// TwinCAT 3 PLC project MAS418
// ProgramVersion: 3.1.4023.0
// libraries:
//   Tc2_Standard, * (Beckhoff Automation GmbH)
//   Tc2_System, * (Beckhoff Automation GmbH)
//   Tc3_Module, * (Beckhoff Automation GmbH)
// project tree:
//   ControlBox/ CL_PC.TcPOU, E_Control_Mode.TcDUT, E_Status.TcDUT, FB_Connect.TcPOU, FB_ControlBox.TcPOU, FB_Encoder.TcPOU, FB_JoystickInputScaling.TcPOU, FB_PathGenerator.TcPOU, FB_Real_Controller.TcPOU, FB_ValveOutput.TcPOU, FB_Virtual_Controller.TcPOU, I_ControlBox.TcIO, OL_VC.TcPOU, ST_Control_Box.TcDUT, ST_ValveDeadBand.TcDUT (not stored)
//   ControlBox/GVL/ G_ControlBox.TcGVL, G_HMI.TcGVL, G_Input.TcGVL (not stored), G_IO_Parameters.TcGVL, G_Output.TcGVL, G_PathGen.TcGVL, G_Sim.TcGVL (not stored)
//   / GlobalTextList.TcGTLO, PlcTask.TcTTO, Visualization Manager.TcVMO (not stored)
//   HMI/ Visualization.TcVIS
//   Programs/FunctionBlock/ FB_Scaling.TcPOU
//   Programs/Functions/ F_NormFlow.TcPOU, F_Scaling.TcPOU, F_Hestunger.TcPOU
//   Programs/ MAIN.TcPOU, P_ControlBox.TcPOU
// real-time tasks:
//   TASK PlcTask: cycle T#10ms, priority 20, ADS port 350
// I/O:
//   DEVICE PLC (disabled), AmsNetId 192.168.56.1.2.1
//     Term 1 (EK1200) [EK1200-5000 EtherCAT Power supply (2A E-Bus)]
//       Term 2 (EL2008-0015) [EL2008-0015 8Ch. Dig. Output 24V DC, 0.35A, not short-circuit proof]
//       Term 3 (EL9011) [EL9011 End Terminal]
//   DEVICE Device 4 (EtherCAT), AmsNetId 5.80.90.242.5.1
//     Term 4 (EK1100) [EK1100 EtherCAT Coupler (2A E-Bus)]
//       DI1 (EL1008) [EL1008 8Ch. Dig. Input 24V, 3ms]
//       DO1 (EL2008)
//       AI1 (EL3068) [EL3068 8Ch. Ana. Input 0-10V]
//       AI2 (EL3068)
//       AI3 ( EL3174)
//       AI4  (EL3255) [EL3255 5Ch. potentiometer measurement with sensor supply]
//       AO1 (EL4104) [EL4104 4Ch. Ana. Output 0-10V, 16bit]
//       Term 10 (EL9011)
//     Encoder [Absolute Rotary Encoder IXARC V01.05]
// variable links:
//   MAS418 Instance <-> Device 4 (EtherCAT)/Encoder
//     PlcTask Inputs/G_Input.n_WinchEncoder <-> Encoder/Position Value
//   MAS418 Instance <-> Device 4 (EtherCAT)/Term 4 (EK1100)/AI1 (EL3068)
//     PlcTask Inputs/G_Input.n_pCA <-> AI Standard Channel 4/Value
//     PlcTask Inputs/G_Input.n_pCB <-> AI Standard Channel 3/Value
//     PlcTask Inputs/G_Input.n_pR <-> AI Standard Channel 2/Value
//     PlcTask Inputs/G_Input.n_pS <-> AI Standard Channel 1/Value
//     PlcTask Inputs/G_Input.n_pWA <-> AI Standard Channel 7/Value
//     PlcTask Inputs/G_Input.n_pWA1 <-> AI Standard Channel 5/Value
//     PlcTask Inputs/G_Input.n_pWB <-> AI Standard Channel 8/Value
//     PlcTask Inputs/G_Input.n_pWB1 <-> AI Standard Channel 6/Value
//   MAS418 Instance <-> Device 4 (EtherCAT)/Term 4 (EK1100)/AI2 (EL3068)
//     PlcTask Inputs/G_Input.n_pWD <-> AI Standard Channel 1/Value
//   MAS418 Instance <-> Device 4 (EtherCAT)/Term 4 (EK1100)/AI3 ( EL3174)
//     PlcTask Inputs/G_Input.n_QW <-> AI Standard Channel 1/Value
//   MAS418 Instance <-> Device 4 (EtherCAT)/Term 4 (EK1100)/AI4  (EL3255)
//     PlcTask Inputs/G_Input.n_JoyX <-> AI Standard Channel 2/Value
//     PlcTask Inputs/G_Input.n_JoyY <-> AI Standard Channel 3/Value
//     PlcTask Inputs/G_Input.n_Xc <-> AI Standard Channel 1/Value
//   MAS418 Instance <-> Device 4 (EtherCAT)/Term 4 (EK1100)/AO1 (EL4104)
//     PlcTask Outputs/G_Output.n_CylValveOut <-> AO Output Channel 2/Analog output
//     PlcTask Outputs/G_Output.n_WinchValveOut <-> AO Output Channel 1/Analog output
//   MAS418 Instance <-> Device 4 (EtherCAT)/Term 4 (EK1100)/DI1 (EL1008)
//     PlcTask Inputs/G_Input.bAuto <-> Channel 2/Input
//     PlcTask Inputs/G_Input.bJoyActive <-> Channel 5/Input
//     PlcTask Inputs/G_Input.bManual <-> Channel 1/Input
//     PlcTask Inputs/G_Input.bStart <-> Channel 3/Input
//     PlcTask Inputs/G_Input.bStop <-> Channel 4/Input
//   MAS418 Instance <-> Device 4 (EtherCAT)/Term 4 (EK1100)/DO1 (EL2008)
//     PlcTask Outputs/G_Output.bEnableCylValve <-> Channel 4/Output
//     PlcTask Outputs/G_Output.bEnableWinchValve <-> Channel 3/Output
//     PlcTask Outputs/G_Output.bGreenLED <-> Channel 1/Output
//     PlcTask Outputs/G_Output.bRedLED <-> Channel 2/Output

CONFIGURATION MAS418
    RESOURCE PLC ON TwinCAT3
        TASK PlcTask(INTERVAL := T#10ms, PRIORITY := 20);
        PROGRAM MAIN WITH PlcTask : MAIN;
    END_RESOURCE
END_CONFIGURATION

// ---- ControlBox/E_Control_Mode.TcDUT
{attribute 'qualified_only'}
{attribute 'strict'}
TYPE E_Control_Mode :
(
	OFF := 0,
	MANUAL := 1,
	AUTO := 2
);
END_TYPE

// ---- ControlBox/E_Status.TcDUT
{attribute 'qualified_only'}
{attribute 'strict'}
TYPE E_Status :
(
	NOTREADY,
	READY,
	STARTING,
	RUNNING,
	STOPPING,
	FAULT
);
END_TYPE

// ---- ControlBox/ST_Control_Box.TcDUT
TYPE ST_Control_Box :
STRUCT
	// Control mode variables
	eMode : E_Control_Mode; // Control mode for the control box
	bAuto : BOOL := FALSE; // Auto control mode input
	bManual : BOOL := FALSE; // Manual control mode input

	// Start/stop variables
	bStart : BOOL := FALSE; // Start button input
	bStop : BOOL := FALSE; // Stop button input

	// Joy variables
	bJoyActive : BOOL; // Activate the joystick boolean (Top switch)
	bJoyNotActive: BOOL; // Inverse logic of JoyActive
	fJoyX : REAL := 0; // Variable for storing the joy value in x direction (Cylinder)
	fJoyY : REAL := 0; // Variable for storing the joy value in y direction (Winch)
END_STRUCT
END_TYPE

// ---- ControlBox/GVL/G_ControlBox.TcGVL
VAR_GLOBAL
	// Global variable for control mode
	eMode : E_Control_Mode := E_Control_Mode.OFF;
	
	// GLobal variable for machine status
	eStatus : E_Status := E_Status.NOTREADY;
	
	// Timer between STARTING -> RUNNING and STOPPING -> NOTREADY
	fbTon : TON := ();
	bStartTimer : BOOL := FALSE;
	bTimerDone : BOOL;
	
	bStart : BOOL := FALSE; // Start button input
	bStop : BOOL := FALSE; // Stop button input
	
	bAuto : BOOL := FALSE; // Auto control mode input
	bManual : BOOL := FALSE; // Manual control mode input
	bOff : BOOL := FALSE; // Off mode
	
	bReady : BOOL := FALSE;
	bStarting : BOOL := FALSE;
	bRunning : BOOL := FALSE;
	bStopping : BOOL := FALSE;
	bFault : BOOL := FALSE;
	
	bJoyActive : BOOL; // Activate the joystick boolean (Top switch)
	bJoyNotActive: BOOL; // Inverse logic of JoyActive
	fJoyX : REAL := G_IO_Parameters.fMaxInputValue/2 + G_IO_Parameters.fMinInputValue/2; // Variable for storing the joy value in x direction (Cylinder)
	fJoyY : REAL := G_IO_Parameters.fMaxInputValue/2 + G_IO_Parameters.fMinInputValue/2; // Variable for storing the joy value in y direction (Winch)
	
	// Normalized values between -1 and 1
	fJoyX_Normalized : LREAL;
	fJoyY_Normalized : LREAL;
	
	// Open-Loop Velocity manual mode
	f_uVFF_winch_manual : LREAL;
	f_uVFF_cyl_manual : LREAL;
	
	// Closed-Loop auto mode
	f_uVFF_winch_auto : LREAL;
	f_uVFF_cyl_auto : LREAL;

	f_uPFB_winch_auto : LREAL;
	f_uPFB_cyl_auto : LREAL;
	
	f_u_winch : LREAL; // Summed winch control signal
	f_u_cyl : LREAL; // Summed cylinder control signal
	
	// Proportional gain
	fPGain : LREAL := 1;
	
	// Position feedback variable
	fPositionFeedback_winch : LREAL := 0;
	fPositionFeedback_cyl : LREAL := 0;
	
	fLimitVal : LREAL := 0.05;
END_VAR

// ---- ControlBox/GVL/G_HMI.TcGVL
VAR_GLOBAL	
	
	// inputs
	f_pS : REAL;
	f_pR : REAL;
	f_pCB : REAL;
	f_pCA : REAL;
	f_pWA1 : REAL;
	f_pWB1 : REAL;
	f_pWA: REAL;
	f_pWB : REAL;
	f_pWD : REAL;
	f_QW : REAL;
	f_Xc : REAL;
	f_JoyX : REAL;
	f_JoyY : REAL;
	f_WinchEncoder : LREAL;
	
END_VAR

// ---- ControlBox/GVL/G_IO_Parameters.TcGVL
{attribute 'qualified_only'}
VAR_GLOBAL
	// Joystick parameters
	fMaxInputValue : REAL := 20509.0;
	fMinInputValue : REAL := 11787.0;
	fNeutralInputValue : REAL := 16175;
	fNeutralDeadband : REAL := 50.0;
	fMaxOutputValue  : REAL := 1.0;
	fMinOutputValue : REAL := -1.0;
	fNeutralOutputValue : REAL := 0.0;
	
	// Deadband
	fPosMax : REAL := 29490.0;
	fPosMin : REAL := 20950.0;
	fNegMin : REAL := 18250.0;
	fNegMax : REAL := 9830.0;
	
	fMaxVel : LREAL := 0.05;
	
	fQmax_winch : LREAL := 60/60000; // L/min
	fQmax_cyl : LREAL := 75/60000; // L/min
END_VAR

// ---- ControlBox/GVL/G_Output.TcGVL
VAR_GLOBAL
	// Boolean outputs
	bGreenLED AT %Q* : BOOL;
	bRedLED AT %Q* : BOOL;
	bEnableWinchValve AT %Q* : BOOL;
	bEnableCylValve AT %Q* : BOOL;
	
	// DINT outputs
	n_WinchValveOut AT %Q* : DINT;
	n_CylValveOut AT %Q* : DINT;
END_VAR

// ---- ControlBox/GVL/G_PathGen.TcGVL
VAR_GLOBAL
	Enable : LREAL;
	x0 :LREAL := 0;  // [m], set at start
	x0_winch : LREAL := 0;
	x0_cyl : LREAL := 0;
	v0 :LREAL := 0; // [m/s], set at start
	Position_SP : LREAL := 0.1+x0; // [m], destination point. needs to set with logic. x + x0
	Velocity_SP : LREAL := 0.05*0.3; // [m/s], desired speed
	t0 : LREAL := 5.5; //[s], time to start ramp
	tRamp : LREAL := 1; // [s] ramp time (rise time)
	tHoldPos : LREAL := 1; // [s], time to stay at position before returning
	tVaiable : TIME := T#0S; // Time rising avfter timer is enabled
	tPT : TIME := T#200S; // Stop time for timer. Nessesery to work
	tQ : BOOL; // Gets true when stop time for timer is reached
	tStart : BOOL := FALSE; // enable to start timer. Rising edge start, falling reset
	fTime : LREAL;
	
	// OUTPUTS:
	fPositionRef : LREAL;
	fVelocityRef : LREAL;
	fTimeTot : LREAL; //Time needed to to the complete path
	fError : LREAL; // Should be changed to a BOOL
// SimulationTime is 
END_VAR

// ---- ControlBox/I_ControlBox.TcIO
INTERFACE I_ControlBox

METHOD Joy_Normalized : REAL
VAR_INPUT
	// Joy X
	fJoyX_raw : LREAL;
	// Joy Y
	fJoyY_raw : LREAL;
	
	// Min/max in/out parameters
	fMin_in : LREAL;
	fMax_in : LREAL;
	fMin_out : REAL;
	fMax_out : LREAL;
END_VAR
VAR_OUTPUT
	fJoyX_normalized : LREAL;
	fJoyY_normalized : LREAL;
END_VAR
END_METHOD

METHOD Mode
END_METHOD

METHOD Status
END_METHOD

END_INTERFACE

// ---- Programs/MAIN.TcPOU
PROGRAM MAIN
VAR
	fbScaling : FB_Scaling;
END_VAR

P_ControlBox(); // Run selected control box mode (virtual or real)
fbScaling();

END_PROGRAM

// ---- Programs/FunctionBlock/FB_Scaling.TcPOU
FUNCTION_BLOCK FB_Scaling
VAR
	fbEncoder : FB_Encoder();
	fbValveOutput : FB_ValveOutput();
END_VAR


//Test OK
F_NormFlow(nInput:= G_Input.n_QW,
	fNormalized => G_HMI.f_QW);

//Preassures
F_Scaling(nInput := G_Input.n_pS,
fMaxValOutput := 400,
fOutput => G_HMI.f_pS);

F_Scaling(nInput := G_Input.n_pR,
fMaxValOutput := 40,
fOutput => G_HMI.f_pR);


F_Scaling(nInput := G_Input.n_pCA,
fMaxValOutput := 400,
fOutput => G_HMI.f_pCA );

F_Scaling(nInput := G_Input.n_pCB,
fMaxValOutput := 400,
fOutput => G_HMI.f_pCB);

F_Scaling(nInput := G_Input.n_pWA1,
fMaxValOutput := 400,
fOutput => G_HMI.f_pWA1 );

F_Scaling(nInput := G_Input.n_pWB1,
fMaxValOutput := 400,
fOutput => G_HMI.f_pWB1);

F_Scaling(nInput := G_Input.n_pWA,
fMaxValOutput := 400,
fOutput => G_HMI.f_pWA);

F_Scaling(nInput := G_Input.n_pWB,
fMaxValOutput := 400,
fOutput => G_HMI.f_pWB);

F_Scaling(nInput := G_Input.n_pWD,
fMaxValOutput := 40,
fOutput => G_HMI.f_pWD);

F_Scaling(nInput := G_Input.n_Xc,
fMaxValOutput := 0.5,
fOutput => G_HMI.f_Xc);

fbEncoder(nRawInput:= G_Input.n_WinchEncoder,
fPosition => G_PathGen.x0_winch);

//fbValveOutput(bEnable:=TRUE, bDeadBandCompOn:=TRUE,
//	stValveDeadBand:= st_ValveDeadBand, fNormalizedInput:=G_ControlBox.f_u_winch, nOutput => G_Output.n_WinchValveOut);

//fbValveOutput(bEnable:=TRUE, bDeadBandCompOn:=TRUE,
//	stValveDeadBand:= st_ValveDeadBand, fNormalizedInput:=G_ControlBox.f_u_cyl, nOutput => G_Output.n_CylValveOut);

F_Hestunger(fInput:=G_ControlBox.f_u_winch, nOut => G_Output.n_WinchValveOut);
F_Hestunger(fInput:=G_ControlBox.f_u_cyl, nOut => G_Output.n_CylValveOut);

END_FUNCTION_BLOCK

// ---- ControlBox/FB_Encoder.TcPOU
FUNCTION_BLOCK FB_Encoder
VAR_INPUT
	nRawInput : UDINT;
END_VAR
VAR_OUTPUT
	fPosition 		: LREAL;
END_VAR
VAR PERSISTENT
	nRounds			: DINT;
	nRawLast 		: DINT;
END_VAR	
VAR
	nInput 		: DINT;
	nTempInputDiff	: DINT;
	nCount 			: DINT;
	nMaxValue30bit 	: DINT :=  1073741823; // 2^30 - 1	
	nThreshold30bit	: DINT := nMaxValue30bit/2;
	fScale16bit		: LREAL := 360.0/65535.0; // 360deg/(2^16 - 1)
	fTempPosition   : LREAL;
END_VAR

// Convert to DINT (same as const values)
nInput := UDINT_TO_DINT(nRawInput);

// Define Encoder Rounds
nTempInputDiff := nInput - nRawLast;
IF (nTempInputDiff > nThreshold30bit) THEN
	nRounds := nRounds - 1;
END_IF

IF (nTempInputDiff < -nThreshold30bit) THEN
	nRounds := nRounds + 1;
END_IF

// Count Encoder Rounds
nCount := nInput + nRounds*nMaxValue30bit;

//Position Output
fPosition := (DINT_TO_LREAL(nCount)*fScale16bit - 17574.8)*PI/180 * 0.475 -2; // [m] -2 FORDI PATHGEN VIRKER IKKE MED STORE TALL FOR SOME REASON

END_FUNCTION_BLOCK

// ---- ControlBox/FB_ValveOutput.TcPOU
FUNCTION_BLOCK FB_ValveOutput
VAR_INPUT
	bEnable 			: BOOL;
	bDeadBandCompOn 	: BOOL;
	stValveDeadBand 	: ST_ValveDeadBand;
	fNormalizedInput 	: LREAL;
END_VAR
VAR_OUTPUT
	bEnableValveOutput : BOOL;
	nOutput : INT; 
END_VAR
VAR
	nOffset 	: INT := 19660;
	nMaxValue	: INT := 29490;
	nMinValue 	: INT :=  9830;
	nTempOutput : INT;
END_VAR

IF	bDeadBandCompOn THEN
	IF fNormalizedInput > 0.0 THEN
		nTempOutput := LREAL_TO_INT(ABS(fNormalizedInput*(stValveDeadBand.fPosMax - stValveDeadBand.fPosMin) + stValveDeadBand.fPosMin));
	ELSIF fNormalizedInput < 0.0 THEN
		nTempOutput := LREAL_TO_INT(ABS(fNormalizedInput*(stValveDeadBand.fNegMax - stValveDeadBand.fNegMin) - stValveDeadBand.fNegMin));
	ELSE
		nTempOutput := nOffset;
	END_IF
ELSE
	IF fNormalizedInput > 0.0 THEN
		nTempOutput := LREAL_TO_INT(ABS(fNormalizedInput*(32767.0 - 19660.0) + 19660.0));
	ELSIF fNormalizedInput < 0.0 THEN
		nTempOutput := LREAL_TO_INT(ABS(fNormalizedInput*(0 - 19660.0) - 19660.0));
	ELSE
		nTempOutput := nOffset;
	END_IF	
END_IF	

IF bEnable THEN
	nOutput := LIMIT(nMinValue, nTempOutput, nMaxValue);
	bEnableValveOutput := TRUE; 
ELSE 	
	nOutput := nOffset;
	bEnableValveOutput := FALSE;	
END_IF

END_FUNCTION_BLOCK

// ---- Programs/Functions/F_NormFlow.TcPOU
FUNCTION F_NormFlow
VAR_INPUT
	nInput : DINT; // 0 to 32767, live data
END_VAR
VAR_OUTPUT
	fNormalized: REAL; // -150 to 150. Scalable by multiplying 
END_VAR
VAR
	fInput : REAL;
	fMAXval : REAL := 32767; //the crayzy guys coming in from the analog input
END_VAR

// TESTE

fInput := DINT_TO_REAL(nInput); 

fNormalized :=  150*(finput-fMaxval/2)/fMaxval*2 + 8.5; // Calibrated by Pers Mekaniske 21.03.23, ISO 301495682 12095 13556478

END_FUNCTION

// ---- Programs/Functions/F_Scaling.TcPOU
FUNCTION F_Scaling
VAR_INPUT
	nInput : DINT; // 0 to 32767, live data
	fMaxValOutput : REAL; // End value for scaling spectrum. EKS: 40 if 0-40 Bar.
END_VAR
VAR_OUTPUT
	fOutput : REAL; // 0 to fMaxValOutput.
END_VAR
VAR
	fInput : REAL;
	fMAXval : REAL := 32767; //the crayzy guys coming in from the analog input
END_VAR

fInput := DINT_TO_REAL(nInput); 

fOutput := fInput/fMAXval*fMaxValOutput;

END_FUNCTION

// ---- Programs/Functions/F_Hestunger.TcPOU
FUNCTION F_Hestunger
VAR_INPUT
	fInput : REAL; // -1 to 1
END_VAR
VAR_OUTPUT
	nOut : DINT;
END_VAR
VAR
	fOutput : REAL; // 0 - 32767 hestunger
END_VAR

fOutput := (fInput+1)/2 * 32767;
nOut := REAL_TO_DINT(fOutput);

END_FUNCTION

// ---- Programs/P_ControlBox.TcPOU
PROGRAM P_ControlBox
VAR
	fbControlBox : FB_ControlBox;
	fbScaling : FB_Scaling;
END_VAR

fbControlBox(bRealControlBox := TRUE); // Run controlbox FB with argument. If bRealControlBox is TRUE, then the FB_RealControlBox will be selected when running the program.
fbScaling();

END_PROGRAM

// ---- ControlBox/FB_ControlBox.TcPOU
FUNCTION_BLOCK FB_ControlBox
VAR_INPUT
	bRealControlBox : BOOL;
END_VAR
VAR_OUTPUT
END_VAR
VAR
	fbVirtualControlBox : FB_Virtual_Controller;
	fbRealControlBox : FB_Real_Controller;
	fbSelectedControlBox : I_ControlBox := fbVirtualControlBox;
	
	// Open Loop velocity control manual mode
	fb_OL_VC_winch_manual : OL_VC;
	fb_OL_VC_cyl_manual : OL_VC;
	
	// Closed Loop position control auto mode
	fb_OL_VC_winch_auto : OL_VC;
	fb_OL_VC_cyl_auto : OL_VC;
	
	fb_CL_PC_winch_auto : CL_PC;
	fb_CL_PC_cyl_auto : CL_PC;
	
	// Path generator
	fbTon : TON;
	fbPathGen : FB_PathGenerator;
	
	fbConnect : FB_Connect;
	fbNormalizeJoyX : FB_JoystickInputScaling;
	fbNormalizeJoyY : FB_JoystickInputScaling;
END_VAR

IF bRealControlBox THEN
	fbSelectedControlBox := fbRealControlBox;
	fbConnect();
ELSE
	fbVirtualControlBox.Sim();
END_IF

// Run mode and status function blocks in selected controlbox
fbSelectedControlBox.Mode();
fbSelectedControlBox.Status();

// Normalize joystick input to -1,1
(*fbSelectedControlBox.Joy_Normalized(fJoyX_raw := G_ControlBox.fJoyX, fJoyY_raw := G_ControlBox.fJoyY,
									fMin_in := G_IO_Parameters.fMinInputValue, fMax_in := G_IO_Parameters.fMaxInputValue,
									fMin_out := G_IO_Parameters.fMinOutputValue, fMax_out := G_IO_Parameters.fMaxOutputValue,
									fJoyX_normalized => G_ControlBox.fJoyX_Normalized, fJoyY_normalized => G_ControlBox.fJoyY_Normalized);
*)	
fbNormalizeJoyX(bEnable:=TRUE, nRawInput:= G_Input.n_JoyX, fNormalizedOutput => G_ControlBox.fJoyX_Normalized);
fbNormalizeJoyY(bEnable:=TRUE, nRawInput:= G_Input.n_JoyY, fNormalizedOutput => G_ControlBox.fJoyY_Normalized);

// Manual mode
// Run Open-Loop control for either winch or cylinder based on input, saturated to -0.05,0.05 m/s					
fb_OL_VC_winch_manual(bEnable:=(G_ControlBox.bRunning AND G_ControlBox.bJoyActive AND G_ControlBox.bManual), 
								fvRef:=G_IO_Parameters.fMaxVel*G_ControlBox.fJoyY_Normalized, 
								fQmax:=G_IO_Parameters.fQmax_winch, 
								f_uVFF => G_ControlBox.f_uVFF_winch_manual);
								
fb_OL_VC_cyl_manual(bEnable:=(G_ControlBox.bRunning AND NOT G_ControlBox.bJoyActive AND G_ControlBox.bManual), 
							  fvRef:=G_IO_Parameters.fMaxVel*G_ControlBox.fJoyX_Normalized, 
							  fQmax:=G_IO_Parameters.fQmax_cyl, 
							  f_uVFF => G_ControlBox.f_uVFF_cyl_manual);

// Auto mode
//Timer for path generator
fbTon(IN := G_PathGen.tStart,
	PT := G_PathGen.tPT,
	Q => G_PathGen.tQ,
	ET => G_PathGen.tVaiable);

G_PathGen.fTime := TIME_TO_LREAL(G_PathGen.tVaiable)/1000;

// Path generator function block
IF G_ControlBox.bJoyActive THEN
fbPathGen(Enable := (G_ControlBox.bAuto AND G_ControlBox.bRunning),
	x0m := G_PathGen.x0_winch,
	v0ms := G_PathGen.v0,
	Position_SPm := G_PathGen.Position_SP,
	Velocity_SPms := G_PathGen.Velocity_SP,
	t0s := G_PathGen.t0,
	tRamps := G_PathGen.tRamp,
	tHoldPoss := G_PathGen.tHoldPos,
	t := G_PathGen.fTime,
	PositionRefm => G_PathGen.fPositionRef,
	VelocityRefms => G_PathGen.fVelocityRef,
	TimeTot => G_PathGen.fTimeTot,
	Error => G_PathGen.fError);
ELSE
fbPathGen(Enable := (G_ControlBox.bAuto AND G_ControlBox.bRunning),
	x0m := G_PathGen.x0,
	v0ms := G_PathGen.v0,
	Position_SPm := G_PathGen.Position_SP,
	Velocity_SPms := G_PathGen.Velocity_SP,
	t0s := G_PathGen.t0,
	tRamps := G_PathGen.tRamp,
	tHoldPoss := G_PathGen.tHoldPos,
	t := G_PathGen.fTime,
	PositionRefm => G_PathGen.fPositionRef,
	VelocityRefms => G_PathGen.fVelocityRef,
	TimeTot => G_PathGen.fTimeTot,
	Error => G_PathGen.fError);
END_IF

// Open-Loop function blocks for winch and cylinder in auto mode
fb_OL_VC_winch_auto(bEnable:=(G_ControlBox.bRunning AND G_ControlBox.bJoyActive AND G_ControlBox.bAuto), 
							  fvRef:=G_PathGen.fVelocityRef, 
							  fQmax:=G_IO_Parameters.fQmax_winch, 
							  f_uVFF => G_ControlBox.f_uVFF_winch_auto);
							  
fb_OL_VC_cyl_auto(bEnable:=(G_ControlBox.bRunning AND NOT G_ControlBox.bJoyActive AND G_ControlBox.bAuto), 
							fvRef:=G_PathGen.fVelocityRef, 
							fQmax:=G_IO_Parameters.fQmax_cyl, 
							f_uVFF => G_ControlBox.f_uVFF_cyl_auto);

// Closed-Loop function blocks for winch ander cylinder in auto mode
fb_CL_PC_winch_auto(bEnable:=(G_ControlBox.bRunning AND G_ControlBox.bJoyActive AND G_ControlBox.bAuto), 
							  fProportionalGain:=G_ControlBox.fPGain, 
							  fPositionReference:=G_PathGen.fPositionRef, 
							  fPositionFeedback:=G_ControlBox.fPositionFeedback_winch, 
							  uPFB => G_ControlBox.f_uPFB_winch_auto);
							  
fb_CL_PC_cyl_auto(bEnable:=(G_ControlBox.bRunning AND NOT G_ControlBox.bJoyActive AND G_ControlBox.bAuto), 
							fProportionalGain:=G_ControlBox.fPGain, 
							fPositionReference:=G_PathGen.fPositionRef, 
							fPositionFeedback:=G_ControlBox.fPositionFeedback_cyl, 
							uPFB => G_ControlBox.f_uPFB_cyl_auto);

// Calculate summed control signals for winch and cylinder
IF G_ControlBox.f_uVFF_winch_auto + G_ControlBox.f_uPFB_winch_auto >= 1 THEN
	G_ControlBox.f_u_winch := 1;
ELSIF G_ControlBox.f_uVFF_winch_auto + G_ControlBox.f_uPFB_winch_auto <= -1 THEN
	G_ControlBox.f_u_winch := -1;
ELSE
	G_ControlBox.f_u_winch := G_ControlBox.f_uVFF_winch_auto + G_ControlBox.f_uPFB_winch_auto + G_ControlBox.f_uVFF_winch_manual + G_ControlBox.f_uVFF_cyl_manual;
END_IF

IF G_ControlBox.f_uVFF_cyl_auto + G_ControlBox.f_uPFB_cyl_auto >= 1 THEN
	G_ControlBox.f_u_cyl := 1;
ELSIF G_ControlBox.f_uVFF_cyl_auto + G_ControlBox.f_uPFB_cyl_auto <= -1 THEN
	G_ControlBox.f_u_cyl := -1;
ELSE
	G_ControlBox.f_u_cyl := G_ControlBox.f_uVFF_cyl_auto + G_ControlBox.f_uPFB_cyl_auto;
END_IF

END_FUNCTION_BLOCK

// ---- ControlBox/FB_Virtual_Controller.TcPOU
FUNCTION_BLOCK FB_Virtual_Controller IMPLEMENTS I_ControlBox
VAR_INPUT
END_VAR
VAR_OUTPUT
END_VAR
VAR
END_VAR

METHOD Joy_Normalized : REAL
VAR_INPUT
	// Joy X
	fJoyX_raw : LREAL;
	// Joy Y
	fJoyY_raw : LREAL;
	
	// Min/max in/out parameters
	fMin_in : LREAL;
	fMax_in : LREAL;
	fMin_out : REAL;
	fMax_out : LREAL;
END_VAR
VAR_OUTPUT
	fJoyX_normalized : LREAL;
	fJoyY_normalized : LREAL;
END_VAR

fJoyX_normalized := (fJoyX_raw - fMin_in) * (fMax_out - fMin_out) / (fMax_in - fMin_in) + fMin_out;
fJoyY_normalized := (fJoyY_raw - fMin_in) * (fMax_out - fMin_out) / (fMax_in - fMin_in) + fMin_out;
END_METHOD

METHOD Mode
// Select control mode (OFF, MANUAL or AUTO) based on three position switch
CASE G_ControlBox.eMode OF
		E_Control_Mode.OFF: // Case OFF
			IF G_ControlBox.bAuto THEN // If switch is in auto position, set control mode to auto
				G_ControlBox.eMode := E_Control_Mode.AUTO;
			ELSIF G_ControlBox.bManual THEN // Else if switch is in manual position, set control mode to manual
				G_ControlBox.eMode := E_Control_Mode.MANUAL;
			ELSE // If none of the conditions above are met, then stay in off mode
				G_ControlBox.eMode := E_Control_Mode.OFF;
			END_IF
		E_Control_Mode.AUTO: // Case AUTO
			IF G_ControlBox.bManual THEN // If switch is in manual mode, then set control mode to manual
				G_ControlBox.eMode := E_Control_Mode.MANUAL;
			ELSIF NOT G_ControlBox.bAuto THEN // If switch is not in auto position (or implicitly not in manual) then set control mode to off
				G_ControlBox.eMode := E_Control_Mode.OFF;
			ELSE // If none of the conditions above are met, then stay in auto mode
				G_ControlBox.eMode := E_Control_Mode.AUTO;
			END_IF
			G_ControlBox.bManual := FALSE; // Reset bManual variable, since we are now in auto mode
		E_Control_Mode.MANUAL: // Case MANUAL
			IF G_ControlBox.bAuto THEN // If switch is in auto position, change the control mode to auto
				G_ControlBox.eMode := E_Control_Mode.AUTO;
			ELSIF NOT G_ControlBox.bManual THEN // If switch is not in manual position (and implicitly not in auto), then set control mode to off
				G_ControlBox.eMode := E_Control_Mode.OFF;
			ELSE // If none of the conditions above are met, then stay in manual mode
				G_ControlBox.eMode := E_Control_Mode.MANUAL;
			END_IF
			G_ControlBox.bAuto := FALSE; // Reset bAuto variable, since we are now in manual mode
END_CASE
END_METHOD

METHOD Sim
VAR_INPUT
END_VAR
// Run sim based on min max restrictions in G_Sim GVL
IF G_ControlBox.eStatus = E_Status.RUNNING AND G_ControlBox.bManual THEN
	IF G_ControlBox.f_uVFF_cyl_manual > 0 AND G_Sim.nX < G_Sim.xMax THEN
		G_Sim.nX := G_Sim.nX+1;
	END_IF
	IF G_ControlBox.f_uVFF_cyl_manual < 0 AND G_Sim.nX > G_Sim.xMin THEN
		G_Sim.nX := G_Sim.nX-1;
	END_IF
	IF G_ControlBox.f_uVFF_winch_manual > 0 AND G_Sim.nY < G_Sim.yMax THEN
		G_Sim.nY := G_Sim.nY+1;
	END_IF
	IF G_ControlBox.f_uVFF_winch_manual < 0 AND G_Sim.nY > G_Sim.yMin THEN
		G_Sim.nY := G_Sim.nY-1;
	END_IF	
END_IF

IF G_ControlBox.eStatus = E_Status.RUNNING AND G_ControlBox.bAuto THEN
	IF G_ControlBox.f_uVFF_cyl_auto > 0 AND G_Sim.nX < G_Sim.xMax THEN
		G_Sim.nX := G_Sim.nX+1;
	END_IF
	IF G_ControlBox.f_uVFF_cyl_auto < 0 AND G_Sim.nX > G_Sim.xMin THEN
		G_Sim.nX := G_Sim.nX-1;
	END_IF
	IF G_ControlBox.f_uVFF_winch_auto > 0 AND G_Sim.nY < G_Sim.yMax THEN
		G_Sim.nY := G_Sim.nY+1;
	END_IF
	IF G_ControlBox.f_uVFF_winch_auto < 0 AND G_Sim.nY > G_Sim.yMin THEN
		G_Sim.nY := G_Sim.nY-1;
	END_IF	
END_IF
END_METHOD

METHOD Status
// Determine machine status based on interaction
CASE G_ControlBox.eStatus OF
	E_Status.NOTREADY: // Case NOTREADY
		IF NOT(G_ControlBox.eMode = E_Control_Mode.OFF) THEN // If either auto or manual mode is selected with the three way switch, then go to ready state
			G_ControlBox.eStatus := E_Status.READY;
		ELSE
			G_ControlBox.eStatus := E_Status.NOTREADY; // If switch is in off mode, then stay in NOTREADY
		END_IF
	E_Status.READY: // Case READY
		IF NOT(G_ControlBox.bAuto OR G_ControlBox.bManual) THEN // If switch is switched back to off, then go to NOTREADY
			G_ControlBox.eStatus := E_Status.NOTREADY;
		ELSE
			G_ControlBox.eStatus := E_Status.READY; // Else stay in READY
		END_IF
		IF	G_ControlBox.bStart THEN // If start button is pressed, then go to STARTING
			G_ControlBox.eStatus := E_Status.STARTING;
		END_IF
	E_Status.STARTING: // Case STARTING
		G_ControlBox.bStartTimer := TRUE;
		G_ControlBox.fbTon(IN:=G_ControlBox.bStartTimer, PT:=T#2S, Q => G_ControlBox.bTimerDone); // Stay in STARTING for 2s
		G_ControlBox.bStartTimer := FALSE;
		IF G_ControlBox.bTimerDone THEN // If timer is done, proceed
			IF G_ControlBox.eMode = E_Control_Mode.MANUAL OR G_ControlBox.eMode = E_Control_Mode.AUTO THEN // If still in manual or auto mode, proceed
				G_ControlBox.eStatus := E_Status.RUNNING;
			ELSE
				G_ControlBox.eStatus := E_Status.STOPPING; // If in off mode, then go to STOPPING
			END_IF
		G_ControlBox.fbTon(IN:=G_ControlBox.bStartTimer, PT:=T#2S, Q => G_ControlBox.bTimerDone); // Reset timer for next time
		END_IF
	E_Status.RUNNING: // Case RUNNING
		G_PathGen.tStart := TRUE;
		G_ControlBox.bRunning := TRUE; // Update variables, used to control lights in HMI
		G_ControlBox.bStopping := FALSE; // Update variables, used to control lights in HMI
		IF G_ControlBox.bStop OR NOT(G_ControlBox.bAuto OR G_ControlBox.bManual) THEN // If stop button is pressed, or switch is in off mode, then go to STOPPING
			G_ControlBox.eStatus := E_Status.STOPPING;
		END_IF
		IF NOT(G_ControlBox.bStart) AND G_ControlBox.bAuto AND (G_ControlBox.bAuto OR G_ControlBox.bManual) THEN // If start button is not held, in auto mode, then go to STOPPING
			G_ControlBox.eStatus := E_Status.STOPPING;
		END_IF
		IF G_ControlBox.bFault THEN // If fault variable is true while RUNNING, then set status to fault
			G_ControlBox.eStatus := E_Status.FAULT;
		END_IF
	E_Status.STOPPING: // Case STOPPING
		G_ControlBox.bRunning := FALSE; // Update variables
		G_ControlBox.bStopping := TRUE; // Update variables
		
		G_ControlBox.bStartTimer := TRUE;
		G_ControlBox.fbTon(IN:=G_ControlBox.bStartTimer, PT:=T#2S, Q => G_ControlBox.bTimerDone,); // Stay in STOPPING for 2s
		G_ControlBox.bStartTimer := FALSE;
		G_ControlBox.bRunning := FALSE;
		IF G_ControlBox.bTimerDone THEN // If timer is done, then go to NOTREADY
			G_ControlBox.eStatus := E_Status.NOTREADY;
			G_ControlBox.fbTon(IN:=G_ControlBox.bStartTimer, PT:=T#2S, Q => G_ControlBox.bTimerDone); // Reset timer for next time
		END_IF
		G_PathGen.tStart := FALSE;
	E_Status.FAULT: // Case FAULT, not used much time on yet.
		IF G_ControlBox.bFault THEN
			G_ControlBox.eStatus := E_Status.FAULT;
			G_ControlBox.bRunning := FALSE;
		ELSE
			G_ControlBox.eStatus := E_Status.NOTREADY;	
		END_IF
END_CASE
END_METHOD

END_FUNCTION_BLOCK

// ---- ControlBox/FB_Real_Controller.TcPOU
FUNCTION_BLOCK FB_Real_Controller IMPLEMENTS I_ControlBox
VAR_INPUT
END_VAR
VAR_OUTPUT
END_VAR
VAR
END_VAR

{warning 'add method implementation '}
METHOD Joy_Normalized : REAL
VAR_INPUT
	// Joy X
	fJoyX_raw : LREAL;
	// Joy Y
	fJoyY_raw : LREAL;
	
	// Min/max in/out parameters
	fMin_in : LREAL;
	fMax_in : LREAL;
	fMin_out : REAL;
	fMax_out : LREAL;
END_VAR
VAR_OUTPUT
	fJoyX_normalized : LREAL;
	fJoyY_normalized : LREAL;
END_VAR

fJoyX_normalized := (fJoyX_raw - fMin_in) * (fMax_out - fMin_out) / (fMax_in - fMin_in) + fMin_out;
fJoyY_normalized := (fJoyY_raw - fMin_in) * (fMax_out - fMin_out) / (fMax_in - fMin_in) + fMin_out;
END_METHOD

METHOD Mode
// Select control mode (OFF, MANUAL or AUTO) based on three position switch
CASE G_ControlBox.eMode OF
		E_Control_Mode.OFF: // Case OFF
			IF G_ControlBox.bAuto THEN // If switch is in auto position, set control mode to auto
				G_ControlBox.eMode := E_Control_Mode.AUTO;
			ELSIF G_ControlBox.bManual THEN // Else if switch is in manual position, set control mode to manual
				G_ControlBox.eMode := E_Control_Mode.MANUAL;
			ELSE // If none of the conditions above are met, then stay in off mode
				G_ControlBox.eMode := E_Control_Mode.OFF;
			END_IF
		E_Control_Mode.AUTO: // Case AUTO
			IF G_ControlBox.bManual THEN // If switch is in manual mode, then set control mode to manual
				G_ControlBox.eMode := E_Control_Mode.MANUAL;
			ELSIF NOT G_ControlBox.bAuto THEN // If switch is not in auto position (or implicitly not in manual) then set control mode to off
				G_ControlBox.eMode := E_Control_Mode.OFF;
			ELSE // If none of the conditions above are met, then stay in auto mode
				G_ControlBox.eMode := E_Control_Mode.AUTO;
			END_IF
			G_ControlBox.bManual := FALSE; // Reset bManual variable, since we are now in auto mode
		E_Control_Mode.MANUAL: // Case MANUAL
			IF G_ControlBox.bAuto THEN // If switch is in auto position, change the control mode to auto
				G_ControlBox.eMode := E_Control_Mode.AUTO;
			ELSIF NOT G_ControlBox.bManual THEN // If switch is not in manual position (and implicitly not in auto), then set control mode to off
				G_ControlBox.eMode := E_Control_Mode.OFF;
			ELSE // If none of the conditions above are met, then stay in manual mode
				G_ControlBox.eMode := E_Control_Mode.MANUAL;
			END_IF
			G_ControlBox.bAuto := FALSE; // Reset bAuto variable, since we are now in manual mode
END_CASE
END_METHOD

METHOD Status
// Determine machine status based on interaction
CASE G_ControlBox.eStatus OF
	E_Status.NOTREADY: // Case NOTREADY
		IF NOT(G_ControlBox.eMode = E_Control_Mode.OFF) THEN // If either auto or manual mode is selected with the three way switch, then go to ready state
			G_ControlBox.eStatus := E_Status.READY;
		ELSE
			G_ControlBox.eStatus := E_Status.NOTREADY; // If switch is in off mode, then stay in NOTREADY
		END_IF
	E_Status.READY: // Case READY
		IF NOT(G_ControlBox.bAuto OR G_ControlBox.bManual) THEN // If switch is switched back to off, then go to NOTREADY
			G_ControlBox.eStatus := E_Status.NOTREADY;
		ELSE
			G_ControlBox.eStatus := E_Status.READY; // Else stay in READY
		END_IF
		IF	G_ControlBox.bStart THEN // If start button is pressed, then go to STARTING
			G_ControlBox.eStatus := E_Status.STARTING;
		END_IF
	E_Status.STARTING: // Case STARTING
		G_PathGen.x0 := G_HMI.f_Xc;
		G_PathGen.Position_SP := 0.1+G_PathGen.x0;
		G_ControlBox.bStartTimer := TRUE;
		G_ControlBox.fbTon(IN:=G_ControlBox.bStartTimer, PT:=T#2S, Q => G_ControlBox.bTimerDone); // Stay in STARTING for 2s
		G_ControlBox.bStartTimer := FALSE;
		IF G_ControlBox.bTimerDone THEN // If timer is done, proceed
			IF G_ControlBox.eMode = E_Control_Mode.MANUAL OR G_ControlBox.eMode = E_Control_Mode.AUTO THEN // If still in manual or auto mode, proceed
				G_ControlBox.eStatus := E_Status.RUNNING;
			ELSE
				G_ControlBox.eStatus := E_Status.STOPPING; // If in off mode, then go to STOPPING
			END_IF
		G_ControlBox.fbTon(IN:=G_ControlBox.bStartTimer, PT:=T#2S, Q => G_ControlBox.bTimerDone); // Reset timer for next time
		END_IF
	E_Status.RUNNING: // Case RUNNING
		G_PathGen.tStart := TRUE;
		G_ControlBox.bRunning := TRUE; // Update variables, used to control lights in HMI
		G_ControlBox.bStopping := FALSE; // Update variables, used to control lights in HMI
		IF G_ControlBox.bStop OR NOT(G_ControlBox.bAuto OR G_ControlBox.bManual) THEN // If stop button is pressed, or switch is in off mode, then go to STOPPING
			G_ControlBox.eStatus := E_Status.STOPPING;
		END_IF
		IF NOT(G_ControlBox.bStart) AND G_ControlBox.bAuto AND (G_ControlBox.bAuto OR G_ControlBox.bManual) THEN // If start button is not held, in auto mode, then go to STOPPING
			G_ControlBox.eStatus := E_Status.STOPPING;
		END_IF
		IF G_ControlBox.bFault THEN // If fault variable is true while RUNNING, then set status to fault
			G_ControlBox.eStatus := E_Status.FAULT;
		END_IF
	E_Status.STOPPING: // Case STOPPING
		G_ControlBox.bRunning := FALSE; // Update variables
		G_ControlBox.bStopping := TRUE; // Update variables
		
		G_ControlBox.bStartTimer := TRUE;
		G_ControlBox.fbTon(IN:=G_ControlBox.bStartTimer, PT:=T#2S, Q => G_ControlBox.bTimerDone,); // Stay in STOPPING for 2s
		G_ControlBox.bStartTimer := FALSE;
		G_ControlBox.bRunning := FALSE;
		IF G_ControlBox.bTimerDone THEN // If timer is done, then go to NOTREADY
			G_ControlBox.eStatus := E_Status.NOTREADY;
			G_ControlBox.fbTon(IN:=G_ControlBox.bStartTimer, PT:=T#2S, Q => G_ControlBox.bTimerDone); // Reset timer for next time
		END_IF
		G_PathGen.tStart := FALSE;
	E_Status.FAULT: // Case FAULT, not used much time on yet.
		IF G_ControlBox.bFault THEN
			G_ControlBox.eStatus := E_Status.FAULT;
			G_ControlBox.bRunning := FALSE;
		ELSE
			G_ControlBox.eStatus := E_Status.NOTREADY;	
		END_IF
END_CASE
END_METHOD

END_FUNCTION_BLOCK

// ---- ControlBox/OL_VC.TcPOU
FUNCTION_BLOCK OL_VC
VAR_INPUT
    bEnable: BOOL; // Enable signal
    fvRef: LREAL; // m/s
    fQmax: LREAL; // L/min
END_VAR
VAR_OUTPUT
    f_uVFF: LREAL; // Output control signal velocity feedforward
END_VAR
VAR_TEMP
    rtb_Q_refm3s: LREAL := 0;
END_VAR

// Open-loop velocity control
IF fvRef > 0.0 THEN 
    rtb_Q_refm3s := 0.0033183 * fvRef;
ELSE 
    rtb_Q_refm3s := fvRef * 0.0023562;
END_IF;

IF bEnable THEN 
    f_uVFF := (60000.0 * rtb_Q_refm3s) / fQmax;
ELSE 
    f_uVFF := 0.0;
END_IF;

END_FUNCTION_BLOCK

// ---- ControlBox/CL_PC.TcPOU
FUNCTION_BLOCK CL_PC
VAR_INPUT
    fProportionalGain: LREAL; // P gain
    fPositionReference: LREAL; // Position ref
    fPositionFeedback: LREAL; // Position feedback
    bEnable: BOOL; // Enable signal
END_VAR
VAR_OUTPUT
    uPFB: LREAL; // Control signal from position feedback loop
    fPositionError: LREAL; // Position error
END_VAR


fPositionError := fPositionReference - fPositionFeedback;
uPFB := fProportionalGain * fPositionError;

IF uPFB > 1.0 THEN 
    uPFB := 1.0;
ELSIF uPFB < -1.0 THEN 
    uPFB := -1.0;
END_IF;

IF NOT bEnable THEN 
    uPFB := 0.0;
END_IF;

END_FUNCTION_BLOCK

// ---- ControlBox/FB_PathGenerator.TcPOU
FUNCTION_BLOCK FB_PathGenerator
VAR_INPUT
    Enable: BOOL;
    x0m: REAL;
    v0ms: LREAL;
    Position_SPm: LREAL;
    Velocity_SPms: LREAL;
    t0s: LREAL;
    tRamps: LREAL;
    tHoldPoss: LREAL;
    t: LREAL;
END_VAR
VAR_OUTPUT
    PositionRefm: LREAL;
    VelocityRefms: LREAL;
    TimeTot: LREAL;
    Error: LREAL;
END_VAR
VAR_TEMP
    Error_0: DINT;
    tHold: LREAL;
    x1: LREAL;
    x4: LREAL;
    a_tmp: LREAL;
    a_tmp_tmp: LREAL;
    a_tmp_0: LREAL;
    a_tmp_tmp_0: LREAL;
    a_tmp_tmp_1: LREAL;
    a_tmp_tmp_2: LREAL;
    x1_tmp: LREAL;
    x4_tmp: LREAL;
END_VAR

(*
 *
 * File: MotionReferenceGeneratorCrane.exp
 *
 * IEC 61131-3 Structured Text (ST) code generated for subsystem "MotionReferenceGeneratorCrane/Subsystem"
 *
 * Model name                      : MotionReferenceGeneratorCrane
 * Model version                   : 1.11
 * Model creator                   : Bruker
 * Model last modified by          : Bruker
 * Model last modified on          : Tue Mar 07 16:29:46 2023
 * Model sample time               : 0.01s
 * Subsystem name                  : MotionReferenceGeneratorCrane/Subsystem
 * Subsystem sample time           : 0.01s
 * Simulink PLC Coder version      : 3.7 (R2022b) 13-May-2022
 * ST code generated on            : Tue Mar 07 16:30:16 2023
 *
 * Target IDE selection            : 3S CoDeSys 2.3
 * Test Bench included             : No
 *
 *)

(* Outputs for Atomic SubSystem: '<Root>/Subsystem' *)
(* MATLAB Function: '<S1>/MATLAB Function' *)
(* MATLAB Function 'Subsystem/MATLAB Function': '<S2>:1' *)
(* '<S2>:1:2' x_SP = x_ref-x0; *)
(* '<S2>:1:3' vs=v_ref; *)
(* '<S2>:1:4' slopeExt = v0-vs; *)
(* '<S2>:1:5' slopeRetr = -vs-v0; *)
(* '<S2>:1:7' as = vs/tRamp; *)
(* '<S2>:1:8' s_acc = (vs^2-v0^2)/as; *)
(* '<S2>:1:10' tHold =(x_SP-s_acc)/vs; *)
tHold := ((Position_SPm - x0m) - (((Velocity_SPms * Velocity_SPms) - (v0ms * v0ms)) / (Velocity_SPms / tRamps))) / Velocity_SPms;
(* '<S2>:1:13' if tHold < 0 *)
IF tHold < 0.0 THEN 
    (* '<S2>:1:14' Error = 1; *)
    Error_0 := 1;
ELSE 
    (* '<S2>:1:15' else *)
    (* '<S2>:1:16' Error = 0; *)
    Error_0 := 0;
END_IF;
(* '<S2>:1:19' t1 = tRamp; *)
(* '<S2>:1:20' t2 = tHold; *)
(* '<S2>:1:21' t3 = tRamp; *)
(* '<S2>:1:22' t4 = tWait; *)
(* '<S2>:1:23' t5 = t1; *)
(* '<S2>:1:24' t6 = t2; *)
(* '<S2>:1:25' t7 = t3; *)
(* '<S2>:1:27' x1 = x0 +v0*((t0+t1)-t0)-(slopeExt/t1)*((t0+t1)-t0)^2/2; *)
a_tmp_tmp := t0s + tRamps;
a_tmp := a_tmp_tmp - t0s;
x1_tmp := (v0ms - Velocity_SPms) / tRamps;
x1 := ((a_tmp * v0ms) + x0m) - ((x1_tmp * (a_tmp * a_tmp)) / 2.0);
(* '<S2>:1:28' x2 = x1 + vs*((t0+t1+t2) -(t0+t1)); *)
(* '<S2>:1:29' x4 = x_ref - v0*((t0+t1+t2+t3+t4+t5)-(t0+t1+t2+t3+t4)) + (slopeRetr/t5)*((t0+t1+t2+t3+t4+t5)-(t0+t1+t2+t3+t4))^2/2; *)
a_tmp_tmp_0 := a_tmp_tmp + tHold;
a_tmp_tmp_1 := a_tmp_tmp_0 + tRamps;
a_tmp := a_tmp_tmp_1 + tHoldPoss;
a_tmp_tmp_2 := a_tmp + tRamps;
a_tmp_0 := a_tmp_tmp_2 - a_tmp;
x4_tmp := (( -Velocity_SPms) - v0ms) / tRamps;
x4 := (Position_SPm - (a_tmp_0 * v0ms)) + ((x4_tmp * (a_tmp_0 * a_tmp_0)) / 2.0);
(* '<S2>:1:30' x5 = x4-vs*((t0+t1+t2+t3+t4+t5+t6) - (t0+t1+t2+t3+t4+t5)); *)
(* '<S2>:1:32' if Error == 1 *)
IF Error_0 = 1 THEN 
    (* '<S2>:1:33' x = x0; *)
    PositionRefm := x0m;
    (* '<S2>:1:34' v = v0; *)
    VelocityRefms := v0ms;
ELSIF (t >= 0.0) AND (t < t0s) THEN 
    (* '<S2>:1:35' elseif t>=0 && t<t0 *)
    (* '<S2>:1:36' x = x0; *)
    PositionRefm := x0m;
    (* '<S2>:1:37' v = v0; *)
    VelocityRefms := v0ms;
ELSIF (t >= t0s) AND (t < a_tmp_tmp) THEN 
    (* '<S2>:1:38' elseif t>=t0 && t<(t0+t1) *)
    (* '<S2>:1:39' x = x0 + v0*(t-t0) - (slopeExt/t1)*(t-t0)^2/2; *)
    a_tmp := t - t0s;
    PositionRefm := ((a_tmp * v0ms) + x0m) - ((x1_tmp * (a_tmp * a_tmp)) / 2.0);
    (* '<S2>:1:40' v = v0-(slopeExt/t1)*(t-t0); *)
    VelocityRefms := v0ms - (x1_tmp * a_tmp);
ELSIF (t >= a_tmp_tmp) AND (t < a_tmp_tmp_0) THEN 
    (* '<S2>:1:41' elseif t>=(t0+t1) && t<(t0+t1+t2) *)
    (* '<S2>:1:42' x = x1 + vs*(t-(t0+t1)); *)
    PositionRefm := ((t - a_tmp_tmp) * Velocity_SPms) + x1;
    (* '<S2>:1:43' v = vs; *)
    VelocityRefms := Velocity_SPms;
ELSIF (t >= a_tmp_tmp_0) AND (t < a_tmp_tmp_1) THEN 
    (* '<S2>:1:44' elseif t>=(t0+t1+t2) && t<(t0+t1+t2+t3) *)
    (* '<S2>:1:45' x = x2 + vs*(t-(t0+t1+t2)) + (slopeExt/t3)*(t-(t0+t1+t2))^2/2; *)
    a_tmp := t - a_tmp_tmp_0;
    PositionRefm := ((((a_tmp_tmp_0 - a_tmp_tmp) * Velocity_SPms) + x1) + (a_tmp * Velocity_SPms)) + ((x1_tmp * (a_tmp * a_tmp)) / 2.0);
    (* IKKE OK *)
    (* '<S2>:1:46' v = vs + (slopeExt/t3)*(t-(t0+t1+t2)); *)
    VelocityRefms := (a_tmp * x1_tmp) + Velocity_SPms;
    (* OK *)
ELSIF (t >= a_tmp_tmp_1) AND (t < a_tmp) THEN 
    (* '<S2>:1:47' elseif t>=(t0+t1+t2+t3) && t<(t0+t1+t2+t3+t4) *)
    (* '<S2>:1:48' x = x_ref; *)
    PositionRefm := Position_SPm;
    (* Ser ok ut *)
    (* '<S2>:1:49' v = v0; *)
    VelocityRefms := v0ms;
ELSIF (t >= a_tmp) AND (t < a_tmp_tmp_2) THEN 
    (* '<S2>:1:50' elseif t>=(t0+t1+t2+t3+t4) && t<(t0+t1+t2+t3+t4+t5) *)
    (* '<S2>:1:51' x = x_ref - v0*(t-(t0+t1+t2+t3+t4)) + (slopeRetr/t5)*(t-(t0+t1+t2+t3+t4))^2/2; *)
    a_tmp := t - a_tmp;
    PositionRefm := (Position_SPm - (a_tmp * v0ms)) + ((x4_tmp * (a_tmp * a_tmp)) / 2.0);
    (* '<S2>:1:52' v = v0 + (slopeRetr/t5)*(t-(t0+t1+t2+t3+t4)); *)
    VelocityRefms := (a_tmp * x4_tmp) + v0ms;
ELSE 
    x1_tmp := a_tmp_tmp_2 + tHold;
    IF (t >= a_tmp_tmp_2) AND (t < x1_tmp) THEN 
        (* '<S2>:1:53' elseif t>=(t0+t1+t2+t3+t4+t5) && t<(t0+t1+t2+t3+t4+t5+t6) *)
        (* '<S2>:1:54' x = x4-vs*(t-(t0+t1+t2+t3+t4+t5)); *)
        PositionRefm := x4 - ((t - a_tmp_tmp_2) * Velocity_SPms);
        (* '<S2>:1:55' v = -vs; *)
        VelocityRefms :=  -Velocity_SPms;
    ELSIF (t >= x1_tmp) AND (t < (x1_tmp + tRamps)) THEN 
        (* '<S2>:1:56' elseif t>=(t0+t1+t2+t3+t4+t5+t6) && t<(t0+t1+t2+t3+t4+t5+t6+t7) *)
        (* '<S2>:1:57' x = x5 - vs*(t-(t0+t1+t2+t3+t4+t5+t6)) - (slopeRetr/t3)*(t-(t0+t1+t2+t3+t4+t5+t6))^2/2; *)
        a_tmp := t - x1_tmp;
        PositionRefm := ((x4 - ((x1_tmp - a_tmp_tmp_2) * Velocity_SPms)) - (a_tmp * Velocity_SPms)) - ((x4_tmp * (a_tmp * a_tmp)) / 2.0);
        (* '<S2>:1:58' v = -vs - (slopeRetr/t3)*(t-(t0+t1+t2+t3+t4+t5+t6)); *)
        VelocityRefms := ( -Velocity_SPms) - (a_tmp * x4_tmp);
    ELSE 
        (* '<S2>:1:59' else *)
        (* '<S2>:1:60' x = x0; *)
        PositionRefm := x0m;
        (* '<S2>:1:61' v = v0; *)
        VelocityRefms := v0ms;
    END_IF;
END_IF;
(* Switch: '<S1>/Switch' incorporates:
 *  Switch: '<S1>/Switch1' *)
(* '<S2>:1:64' T = t0+t1+t2+t3+t4+t5+t6+t7; *)
IF NOT Enable THEN 
    (* Outport: '<Root>/PositionRef [m]' *)
//    PositionRefm := 0;
    (* Outport: '<Root>/VelocityRef [m//s]' *)
    VelocityRefms := 0;
END_IF;
(* End of Switch: '<S1>/Switch' *)
(* Outport: '<Root>/TimeTot' incorporates:
 *  MATLAB Function: '<S1>/MATLAB Function' *)
TimeTot := ((((((t0s + tRamps) + tHold) + tRamps) + tHoldPoss) + tRamps) + tHold) + tRamps;
(* Outport: '<Root>/Error' incorporates:
 *  MATLAB Function: '<S1>/MATLAB Function' *)
Error := DINT_TO_LREAL(Error_0);
(* End of Outputs for SubSystem: '<Root>/Subsystem' *)

END_FUNCTION_BLOCK

// ---- ControlBox/FB_Connect.TcPOU
FUNCTION_BLOCK FB_Connect
VAR_INPUT
END_VAR
VAR_OUTPUT
END_VAR
VAR
END_VAR


// INPUTS

// Connect bools
G_ControlBox.bManual := G_Input.bManual;
G_ControlBox.bAuto := G_Input.bAuto;
G_ControlBox.bStart := G_Input.bStart;
G_ControlBox.bStop := G_Input.bStop;
G_ControlBox.bJoyActive := G_Input.bJoyActive;

// Connect winch and cylinder encoders for position feedback
G_ControlBox.fPositionFeedback_winch := G_HMI.f_WinchEncoder;
G_ControlBox.fPositionFeedback_cyl := G_HMI.f_Xc;

// OUTPUTS

// Connect bools
G_Output.bGreenLED := G_ControlBox.bRunning;
G_Output.bRedLED := G_ControlBox.bStopping;
G_Output.bEnableWinchValve := TRUE;
G_Output.bEnableCylValve := TRUE;

// Connect DINTs

END_FUNCTION_BLOCK

// ---- ControlBox/FB_JoystickInputScaling.TcPOU
FUNCTION_BLOCK FB_JoystickInputScaling
VAR_INPUT
	bEnable 				: BOOL;
	nRawInput 				: DINT;
END_VAR
VAR_OUTPUT
	fNormalizedOutput 		: LREAL;
END_VAR
VAR
	fRawInput 				: LREAL;
	fTempInput 				: LREAL;
	fTempOutput 			: LREAL;
END_VAR

fRawInput := DINT_TO_LREAL(nRawInput);

fTempInput := fRawInput - G_IO_Parameters.fNeutralInputValue;

IF fTempInput > G_IO_Parameters.fNeutralDeadband THEN
	fTempOutput := fTempInput/(G_IO_Parameters.fMaxInputValue - G_IO_Parameters.fNeutralInputValue);
ELSIF fTempInput < -G_IO_Parameters.fNeutralDeadband THEN	
	fTempOutput := fTempInput/(G_IO_Parameters.fNeutralInputValue - G_IO_Parameters.fMinInputValue);
ELSE
	fTempOutput := 0.0;
END_IF

IF NOT(bEnable) THEN
	fNormalizedOutput := 0.0;
ELSE
	fNormalizedOutput := LIMIT(G_IO_Parameters.fMinOutputValue, fTempOutput, G_IO_Parameters.fMaxOutputValue);
END_IF

END_FUNCTION_BLOCK

// ---- GlobalTextList.TcGTLO
TEXTLIST GlobalTextList
  175 = '%2.1f m'
  136 = '%2.2f m'
  887 = '%2.3f m'
  961 = '%3.1f bar'
  821 = '%3.1f l/min'
  344 = '%f'
  126 = '%s'
  129 = '+'
  960 = '-'
  818 = 'AUTO'
  514 = 'Cylinder piston'
  233 = 'Cylinder pos'
  927 = 'Cylinder rod'
  139 = 'Flow:'
  914 = 'Joy top switch'
  836 = 'Joy X'
  464 = 'Joy Y'
  149 = 'Load height'
  236 = 'MANUAL'
  890 = 'Mode:'
  417 = 'Position:'
  362 = 'Pressures:'
  985 = 'Return '
  833 = 'Start'
  776 = 'Status:'
  326 = 'Stop'
  60 = 'Supply'
  659 = 'Winch drain'
  85 = 'Winch flow'
  319 = 'Winch in'
  712 = 'Winch in before'
  976 = 'Winch out'
  229 = 'Winch out red'
  907 = 'X:'
  335 = 'Y:'
END_TEXTLIST

// ---- HMI/Visualization.TcVIS
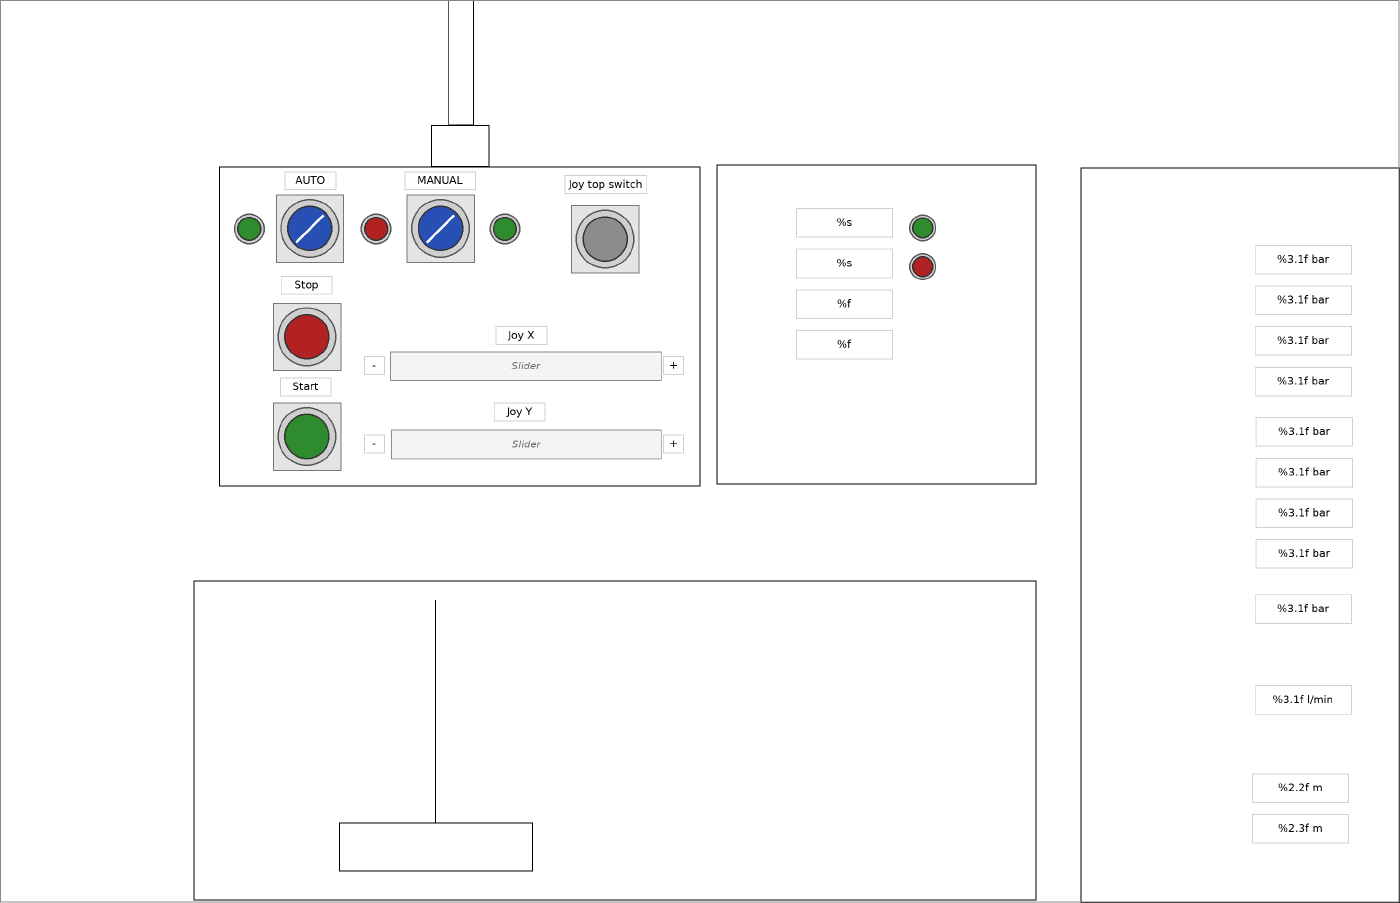
VISUALIZATION Visualization  // 1446x933
    RoundedRectangle (226,172 497x330)
    RotarySwitch (285,201 70x70), variable: G_ControlBox.bAuto, behaviour: TOGGLE, style: Switch-RotarySwitch-Blue
    PushSwitch (282,416 70x70), variable: G_ControlBox.bStart, behaviour: TAP, style: Switch-PushSwitch-Green
    PushSwitch (282,313 70x70), variable: G_ControlBox.bStop, behaviour: TAP, style: Switch-PushSwitch-Red
    RotarySwitch (420,201 70x70), variable: G_ControlBox.bManual, behaviour: TOGGLE, style: Switch-RotarySwitch-Blue
    Slider (404,444 279x30), variable: G_ControlBox.fJoyY, input disabled if: G_ControlBox.bJoyNotActive, scale 0..0
    Slider (403,363 280x30), variable: G_ControlBox.fJoyX, input disabled if: G_ControlBox.bJoyNotActive, scale 0..0
    Rectangle (445,129 60x43)
    Rectangle (463,0 26x129)
    Textfield (290,285 53x19), "Stop"
    Textfield (289,390 53x19), "Start"
    Textfield (512,337 53x19), "Joy X"
    Textfield (510,416 53x19), "Joy Y"
    Textfield (583,181 85x19), "Joy top switch"
    Textfield (685,368 21x19), "+"
    Textfield (685,449 21x19), "+"
    Textfield (376,449 21x19), "-"
    Textfield (376,368 21x19), "-"
    Textfield (294,177 53x19), "AUTO"
    Textfield (418,177 73x19), "MANUAL"
    RoundedRectangle (740,170 330x330)
    Label (756,214 63x30), "Mode:"
    Label (738,253 90x38), "Status:"
    Textfield (822,215 100x30), "%s", text variable: G_ControlBox.eMode
    Lamp1 (937,215 32x41), variable: G_ControlBox.bRunning, style: Lamp-Lamp1-Green
    Textfield (822,257 100x30), "%s", text variable: G_ControlBox.eStatus
    Lamp1 (937,255 32x41), variable: G_ControlBox.bStopping, style: Lamp-Lamp1-Red
    Lamp1 (239,216 37x41), variable: G_ControlBox.bAuto, style: Lamp-Lamp1-Green
    Lamp1 (370,216 37x41), variable: G_ControlBox.bFault, style: Lamp-Lamp1-Red
    Lamp1 (503,216 37x41), variable: G_ControlBox.bManual, style: Lamp-Lamp1-Green
    Textfield (822,299 100x30), "%f", text variable: G_ControlBox.fJoyX_Normalized
    Textfield (822,341 100x30), "%f", text variable: G_ControlBox.fJoyY_Normalized
    Label (780,298 45x38), "X:"
    Label (780,337 45x38), "Y:"
    RoundedRectangle (200,600 870x330)
    Rectangle (350,850 200x50)
        p3528305787: G_Sim.nX
        p2773130477: G_Sim.nY
        p874137650: G_Sim.nX
        p1126004900: G_Sim.nY
    Line (450,850) (450,620)
        p3528305787: G_Sim.nX
        p874137650: G_Sim.nX
        p2773130477: G_Sim.nY
    PushSwitchLed (590,212 70x70), variable: G_ControlBox.bJoyActive, behaviour: TOGGLE, style: Switch-PushSwitchLed-Gray
    RoundedRectangle (1116,173 330x760)
    Label (1205,252 88x30), "Supply"
    Label (1200,291 102x38), "Return"
    Textfield (1296,253 100x30), "%3.1f bar", text variable: G_HMI.f_pS
    Textfield (1296,295 100x30), "%3.1f bar", text variable: G_HMI.f_pR
    Textfield (1296,337 100x30), "%3.1f bar", text variable: G_HMI.f_pCA
    Textfield (1296,379 100x30), "%3.1f bar", text variable: G_HMI.f_pCB
    Label (1156,336 143x38), "Cylinder rod"
    Label (1137,375 162x38), "Cylinder piston"
    Label (1193,430 101x30), "Winch in"
    Label (1123,469 180x38), "Winch in before"
    Textfield (1297,431 100x30), "%3.1f bar", text variable: G_HMI.f_pWA
    Textfield (1297,473 100x30), "%3.1f bar", text variable: G_HMI.f_pWA1
    Textfield (1297,515 100x30), "%3.1f bar", text variable: G_HMI.f_pWA1
    Textfield (1297,557 100x30), "%3.1f bar", text variable: G_HMI.f_pWB
    Label (1176,514 124x38), "Winch out"
    Label (1141,553 159x38), "Winch out red"
    Label (1164,613 129x30), "Winch drain"
    Label (1163,704 139x38), "Winch flow"
    Textfield (1296,614 100x30), "%3.1f bar", text variable: G_HMI.f_pWD
    Textfield (1296,708 100x30), "%3.1f l/min", text variable: G_HMI.f_QW
    Textfield (1293,799 100x30), "%2.2f m", text variable: G_HMI.f_Xc
    Textfield (1293,841 100x30), "%2.3f m", text variable: G_PathGen.x0_winch
    Label (1156,798 140x38), "Cylinder pos"
    Label (1155,837 141x38), "Load height"
    Label (1145,198 194x38), "Pressures:"
    Label (1087,750 251x38), "Position:"
    Label (1065,660 251x38), "Flow:"
END_VISUALIZATION
